FUNCTION_BLOCK INTERNAL FB_State4 EXTENDS FB_State
VAR_INPUT
END_VAR
VAR_OUTPUT
END_VAR
VAR
END_VAR

END_FUNCTION_BLOCK

(* stored: Version 1.1.0.1, ProductVersion 3.1.4024.12
   POU FB_State4: Id {f2d6db61-3f74-0140-1697-2b4311c6a948}, SpecialFunc None *)
